TYPE ST_TopElement2_HMI :
STRUCT
	bZmienneTypoweDlaTopElement2	: BOOL;
	
END_STRUCT
END_TYPE

(* stored: Version 1.1.0.1, ProductVersion 3.1.4024.15
   DUT ST_TopElement2_HMI: Id {9a343522-6a11-420b-8d20-f52071dc6f00} *)
